// SIMATIC S7-200 project (STEP 7-Micro/WIN), CPU 221 REL 01.10

SYMBOL_TABLE USER1
s1               I0.0     // mo thuan
s2               I0.1     // mo nghich
y1               Q0.0     // quay thuan
y2               Q0.1     // quay nghich
s3               I0.2     // stop 1
s4               I0.3     // stop 2
s5               I0.4     // stop 1,2
END_SYMBOL_TABLE

ORGANIZATION_BLOCK MAIN:OB1
TITLE=PROGRAM COMMENTS
BEGIN
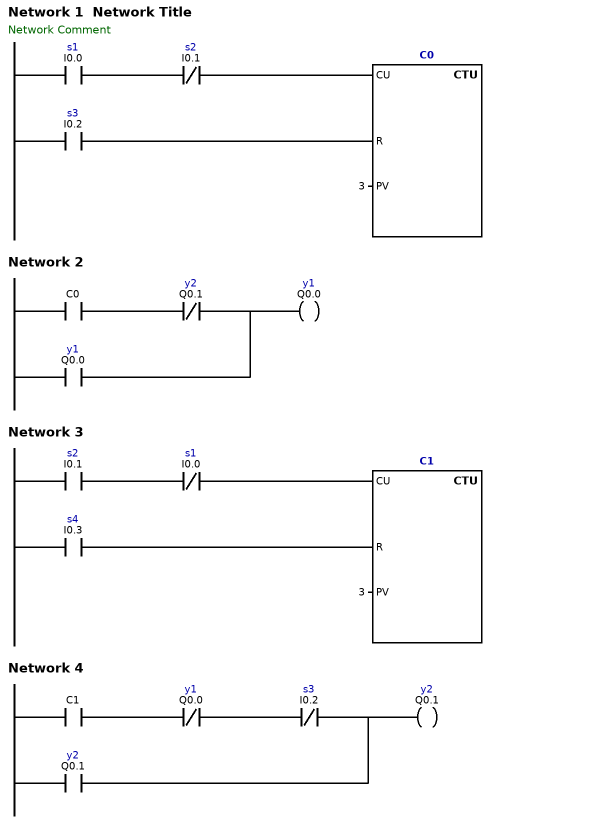
Network 1 // Network Title
// Network Comment
LD     s1:I0.0
AN     s2:I0.1
LD     s3:I0.2
CTU    C0, 3
Network 2
LD     C0
AN     y2:Q0.1
O      y1:Q0.0
=      y1:Q0.0
Network 3
LD     s2:I0.1
AN     s1:I0.0
LD     s4:I0.3
CTU    C1, 3
Network 4
LD     C1
AN     y1:Q0.0
AN     s3:I0.2
O      y2:Q0.1
=      y2:Q0.1
END_ORGANIZATION_BLOCK
